{attribute 'enable_dynamic_creation'}	
{attribute 'no_explicit_call' := 'do not call this function block directly'} 
FUNCTION_BLOCK FileMovePointerTask EXTENDS FileContentTask
VAR
	_ClassName : STRING := __POUNAME();

    _MovePointer : Tc2_System.FB_FileSeek;
END_VAR

{attribute 'monitoring' := 'call'}
PROPERTY ClassName : STRING
GET
ClassName := _ClassName;
END_GET
END_PROPERTY

METHOD Execute : BOOL
VAR_INPUT
	start : BOOL;
END_VAR
IF start THEN
	Validate();

	_MovePointer(
		bExecute := FALSE,
		hFile := FilecontentManager.FileHandle,
		sNetId := FilecontentManager.AmsNetId,
		tTimeout := Timeout
	);	
END_IF

_MovePointer(bExecute := TRUE);

IF _MovePointer.bError THEN
	//exceptionFactory.ThrowException(__POSITION(), WStringHelper.Concat2("Move file pointer failed", GetErrorMessageByErrorId(_MovePointer.nErrId)), __POUNAME(), ClassName, CurrentNamespace.Name, __POSITION(), _MovePointer.nErrId);
ELSIF NOT _MovePointer.bBusy THEN
	Execute := EXECUTION_STATE.DONE;
END_IF
END_METHOD

PROPERTY MovePointerType : FILE_MOVE_POINTER_TYPE
GET
VAR
	resultAddress : POINTER TO INT;
END_VAR
resultAddress := ADR(MovePointerType);
resultAddress^ := _MovePointer.eOrigin;
END_GET
SET
_MovePointer.eOrigin := TO_INT(MovePointerType);
END_SET
END_PROPERTY

PROPERTY NewFilePointerPosition : DINT
GET
NewFilePointerPosition := _MovePointer.nSeekPos;
END_GET
SET
_MovePointer.nSeekPos := NewFilePointerPosition;
END_SET
END_PROPERTY

END_FUNCTION_BLOCK

(* stored: Version 1.1.0.1
   POU FileMovePointerTask: Id {0d6ca812-533d-4e1a-945f-85a946bb861c}, SpecialFunc None
   Property ClassName: Id {0fecaf7d-2316-48d1-947a-0b6e119d32f3}
   Get Get: Id {a8aee7d5-d13c-45f1-93b2-ea1f016cb0e2}
   Method Execute: Id {fdfa44cb-ccec-43d0-8996-4990e338235c}
   Property MovePointerType: Id {e77ee437-6b55-484c-9787-a26f82edbd34}
   Get Get: Id {e35160bc-e62c-4b80-9331-2d52eb54bde3}
   Set Set: Id {aa6d6362-9424-4867-992d-00fa0b72b49d}
   Property NewFilePointerPosition: Id {7772fd5a-ecc0-451c-aae6-229d9ebc1e3b}
   Get Get: Id {faca5697-768d-4e89-86aa-3a433f378ce6}
   Set Set: Id {f0bb5c9b-e478-4a8e-8ae5-41597d402efd} *)
